PROGRAM Measurement_Angle
VAR
    //Feedback calculated in Detector Arc Radius prog
END_VAR

GVL.astAxes[AXIS_MEASUREMENT_ANGLE].stInputs.bLimitBwd := TRUE;
GVL.astAxes[AXIS_MEASUREMENT_ANGLE].stInputs.bLimitFwd := TRUE;
//GVL.astAxes[AXIS_MEASUREMENT_ANGLE].stControl.bEnable := TRUE;

END_PROGRAM

(* stored: Version 1.1.0.1, ProductVersion 3.1.4024.11
   POU Measurement_Angle: Id {f6b3ee24-c778-4988-80a4-3877a9d9ce34}, SpecialFunc None *)
